// TIA Portal V17 export
// export: Created 2024-09-02T12:50:40.0105862Z, ExportSetting WithDefaults, DisplayName Totally Integrated Automation Portal, DisplayVersion V17, DisplayName TIA Portal Openness, DisplayVersion V17, DisplayName TIA Portal Version Control Interface, DisplayVersion V17, DisplayName STEP 7 Professional, DisplayVersion V17, DisplayName STEP 7 Safety, DisplayVersion V17, DisplayName WinCC Professional, DisplayVersion V17
TYPE "Scania_typ_Process"
// stored: IsFailsafeCompliant false
   STRUCT
      StationOperationStatus : "Scania_typ_Status";
      "Program Station" { S7_SetPoint := 'True'} : Int;
      OperationSelection : Array[1..16] of Bool;
      OperationProgram : Array[1..16] of Byte;
      Reserve : Array[1..28] of Byte;
   END_STRUCT;
END_TYPE
